SYSTEM TRAFFIC (* System Configuration *)
  (* Standard: 61499-1 *)
  (* Version 0.4, 2009-03-05, JHC, Holobloc Inc., Deleted Application. *)
  (* Version 0.3, 2003-12-05, JHC, Rockwell Automation, Renamed from NEWSYSTEM. *)
  (* Version 0.2, 2002-11-05, JHC, Rockwell Automation, Fixed missing (empty) FBD in Application. *)
  (* Version 0.1, 2002-01-17, JHC, Rockwell Automation, Minor cleanup *)
  (* Version 0.0, 2000-05-27, JHC, Rockwell Automation *)
  DEVICE Device1 : FRAME_DEVICE(BOUNDS := [100,100,300,110])
    RESOURCE Model : PANEL_RESOURCE
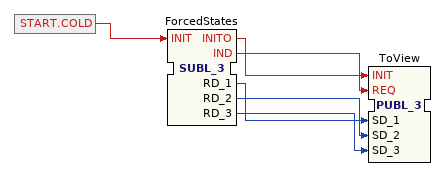
      FBS
        ForcedStates : SUBL_3;
        ToView : PUBL_3;
      END_FBS
      EVENT_CONNECTIONS
        START.COLD TO ForcedStates.INIT;
        ForcedStates.INITO TO ToView.INIT;
        ForcedStates.IND TO ToView.REQ;
      END_CONNECTIONS
      DATA_CONNECTIONS
        ForcedStates.RD_1 TO ToView.SD_1;
        ForcedStates.RD_2 TO ToView.SD_2;
        ForcedStates.RD_3 TO ToView.SD_3;
      END_CONNECTIONS
    END_RESOURCE
    RESOURCE Control : PANEL_RESOURCE
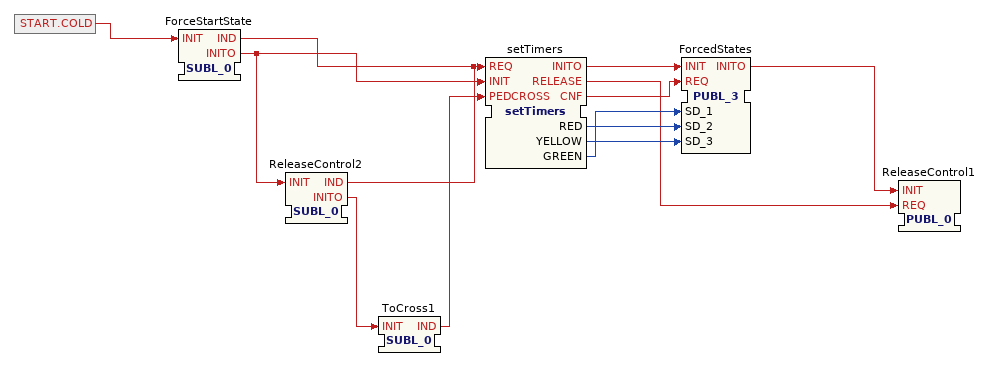
      FBS
        ForcedStates : PUBL_3;
        ForceStartState : SUBL_0;
        setTimers : setTimers;
        ReleaseControl1 : PUBL_0;
        ReleaseControl2 : SUBL_0;
        ToCross1 : SUBL_0;
      END_FBS
      EVENT_CONNECTIONS
        START.COLD TO ForceStartState.INIT;
        setTimers.INITO TO ForcedStates.INIT;
        ForceStartState.IND TO setTimers.REQ;
        ForceStartState.INITO TO setTimers.INIT;
        ForcedStates.INITO TO ReleaseControl1.INIT;
        setTimers.RELEASE TO ReleaseControl1.REQ;
        setTimers.CNF TO ForcedStates.REQ;
        ForceStartState.INITO TO ReleaseControl2.INIT;
        ReleaseControl2.IND TO setTimers.REQ;
        ReleaseControl2.INITO TO ToCross1.INIT;
        ToCross1.IND TO setTimers.PEDCROSS;
      END_CONNECTIONS
      DATA_CONNECTIONS
        setTimers.RED TO ForcedStates.SD_1;
        setTimers.YELLOW TO ForcedStates.SD_2;
        setTimers.GREEN TO ForcedStates.SD_3;
      END_CONNECTIONS
    END_RESOURCE
    RESOURCE View : PANEL_RESOURCE
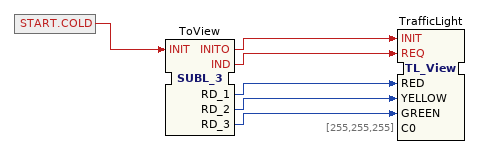
      FBS
        TrafficLight : TL_View(C0 := [255,255,255]);
        ToView : SUBL_3;
      END_FBS
      EVENT_CONNECTIONS
        START.COLD TO ToView.INIT;
        ToView.INITO TO TrafficLight.INIT;
        ToView.IND TO TrafficLight.REQ;
      END_CONNECTIONS
      DATA_CONNECTIONS
        ToView.RD_1 TO TrafficLight.RED;
        ToView.RD_2 TO TrafficLight.YELLOW;
        ToView.RD_3 TO TrafficLight.GREEN;
      END_CONNECTIONS
    END_RESOURCE
    RESOURCE HMI : PANEL_RESOURCE
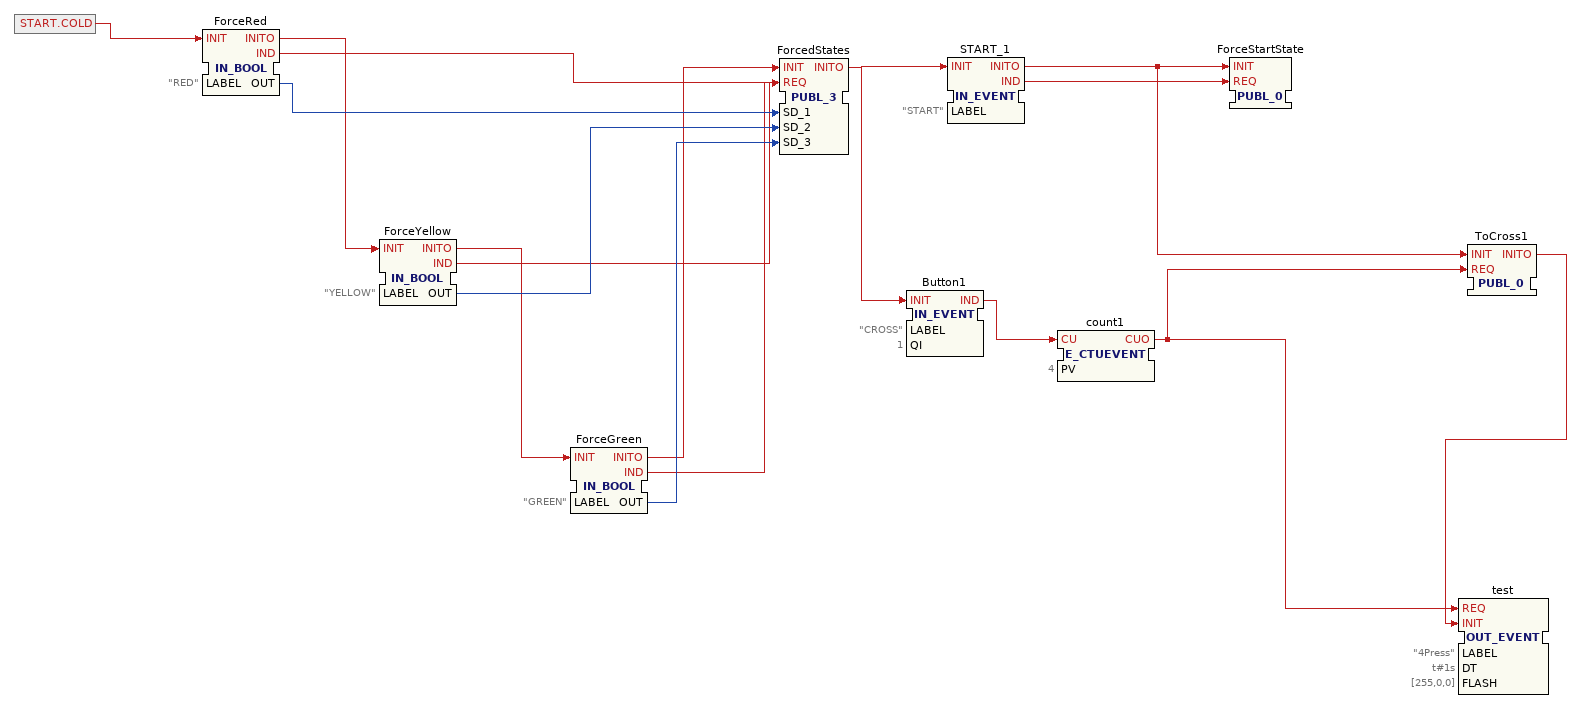
      FBS
        ForceRed : IN_BOOL(LABEL := "RED");
        ForcedStates : PUBL_3;
        ForceYellow : IN_BOOL(LABEL := "YELLOW");
        ForceGreen : IN_BOOL(LABEL := "GREEN");
        START_1 : IN_EVENT(LABEL := "START");
        ForceStartState : PUBL_0;
        Button1 : IN_EVENT(LABEL := "CROSS", QI := 1);
        ToCross1 : PUBL_0;
        count1 : E_CTUEVENT(PV := 4);
        test : OUT_EVENT(LABEL := "4Press", DT := t#1s, FLASH := [255,0,0]);
      END_FBS
      EVENT_CONNECTIONS
        START.COLD TO ForceRed.INIT;
        ForceRed.INITO TO ForceYellow.INIT;
        ForceYellow.INITO TO ForceGreen.INIT;
        ForceGreen.INITO TO ForcedStates.INIT;
        ForceRed.IND TO ForcedStates.REQ;
        ForceYellow.IND TO ForcedStates.REQ;
        ForceGreen.IND TO ForcedStates.REQ;
        ForcedStates.INITO TO START_1.INIT;
        START_1.INITO TO ForceStartState.INIT;
        START_1.IND TO ForceStartState.REQ;
        ForcedStates.INITO TO Button1.INIT;
        START_1.INITO TO ToCross1.INIT;
        Button1.IND TO count1.CU;
        count1.CUO TO ToCross1.REQ;
        count1.CUO TO test.REQ;
        ToCross1.INITO TO test.INIT;
      END_CONNECTIONS
      DATA_CONNECTIONS
        ForceRed.OUT TO ForcedStates.SD_1;
        ForceYellow.OUT TO ForcedStates.SD_2;
        ForceGreen.OUT TO ForcedStates.SD_3;
      END_CONNECTIONS
    END_RESOURCE
  END_DEVICE
  DEVICE Device2 : FRAME_DEVICE(BOUNDS := [100,210,200,110])
    RESOURCE Model : PANEL_RESOURCE
    END_RESOURCE
    RESOURCE Control : PANEL_RESOURCE
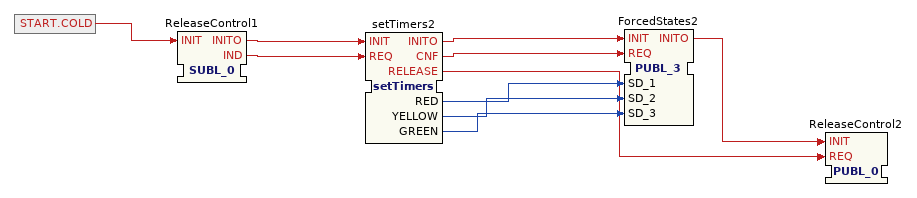
      FBS
        ForcedStates2 : PUBL_3;
        setTimers2 : setTimers;
        ReleaseControl2 : PUBL_0;
        ReleaseControl1 : SUBL_0;
      END_FBS
      EVENT_CONNECTIONS
        setTimers2.INITO TO ForcedStates2.INIT;
        setTimers2.CNF TO ForcedStates2.REQ;
        ForcedStates2.INITO TO ReleaseControl2.INIT;
        START.COLD TO ReleaseControl1.INIT;
        ReleaseControl1.INITO TO setTimers2.INIT;
        ReleaseControl1.IND TO setTimers2.REQ;
        setTimers2.RELEASE TO ReleaseControl2.REQ;
      END_CONNECTIONS
      DATA_CONNECTIONS
        setTimers2.RED TO ForcedStates2.SD_1;
        setTimers2.YELLOW TO ForcedStates2.SD_2;
        setTimers2.GREEN TO ForcedStates2.SD_3;
      END_CONNECTIONS
    END_RESOURCE
    RESOURCE View : PANEL_RESOURCE
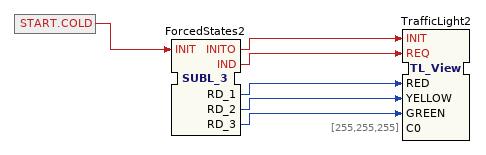
      FBS
        TrafficLight2 : TL_View(C0 := [255,255,255]);
        ForcedStates2 : SUBL_3;
      END_FBS
      EVENT_CONNECTIONS
        START.COLD TO ForcedStates2.INIT;
        ForcedStates2.INITO TO TrafficLight2.INIT;
        ForcedStates2.IND TO TrafficLight2.REQ;
      END_CONNECTIONS
      DATA_CONNECTIONS
        ForcedStates2.RD_1 TO TrafficLight2.RED;
        ForcedStates2.RD_2 TO TrafficLight2.YELLOW;
        ForcedStates2.RD_3 TO TrafficLight2.GREEN;
      END_CONNECTIONS
    END_RESOURCE
    RESOURCE HMI : PANEL_RESOURCE
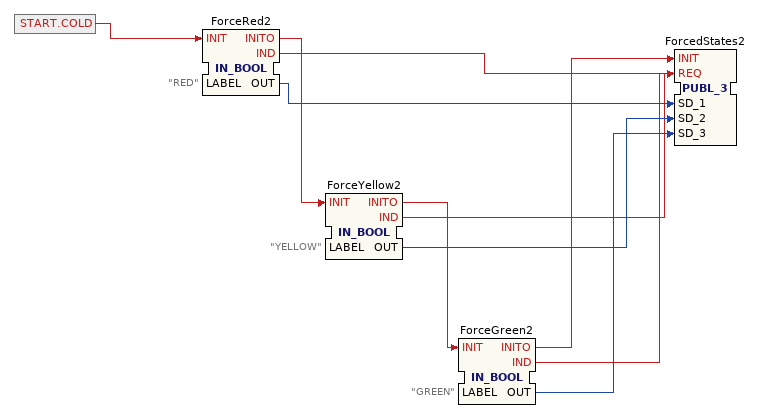
      FBS
        ForceRed2 : IN_BOOL(LABEL := "RED");
        ForcedStates2 : PUBL_3;
        ForceYellow2 : IN_BOOL(LABEL := "YELLOW");
        ForceGreen2 : IN_BOOL(LABEL := "GREEN");
      END_FBS
      EVENT_CONNECTIONS
        START.COLD TO ForceRed2.INIT;
        ForceRed2.INITO TO ForceYellow2.INIT;
        ForceYellow2.INITO TO ForceGreen2.INIT;
        ForceGreen2.INITO TO ForcedStates2.INIT;
        ForceRed2.IND TO ForcedStates2.REQ;
        ForceYellow2.IND TO ForcedStates2.REQ;
        ForceGreen2.IND TO ForcedStates2.REQ;
      END_CONNECTIONS
      DATA_CONNECTIONS
        ForceRed2.OUT TO ForcedStates2.SD_1;
        ForceYellow2.OUT TO ForcedStates2.SD_2;
        ForceGreen2.OUT TO ForcedStates2.SD_3;
      END_CONNECTIONS
    END_RESOURCE
  END_DEVICE
END_SYSTEM
